// TwinCAT 3 PLC project ConveyorBelt
// ProgramVersion: 3.1.4022.3
// libraries:
//   Tc2_Standard, * (Beckhoff Automation GmbH)
//   Tc2_System, * (Beckhoff Automation GmbH)
//   Tc3_Module, * (Beckhoff Automation GmbH)
// project tree:
//   / PlcTask.TcTTO
//   POUs/ MAIN.TcPOU
// real-time tasks:
//   TASK PlcTask: cycle T#10ms, priority 20, ADS port 350

CONFIGURATION ConveyorBelt
    RESOURCE PLC ON TwinCAT3
        TASK PlcTask(INTERVAL := T#10ms, PRIORITY := 20);
        PROGRAM MAIN WITH PlcTask : MAIN;
    END_RESOURCE
END_CONFIGURATION

// ---- POUs/MAIN.TcPOU
PROGRAM MAIN
VAR
END_VAR

VAR_INPUT
	ElevatorSensor AT %IX1.0: BOOL;
	Conveyor2Sensor AT %IX2.0: BOOL;
END_VAR

VAR_OUTPUT
	// Conveyor 1 variables
	Conveyor1 AT %QX0.0: BOOL;
	
	// Elevator variables
	ElevatorConveyor AT %QX1.0: BOOL;
	ElevatorTableUp AT %QX1.1: BOOL;
	ElevatorTableDown AT %QX1.2: BOOL;
	
	// Conveyor 2 variables
	Conveyor2 AT %QX2.0: BOOL;
	PusherPush AT %QX2.1: BOOL;
	PusherReset AT %QX2.2: BOOL;
	
	// Box variables
	BoxShaker AT %QX3.0: BOOL;
END_VAR

END_PROGRAM
